FUNCTION_BLOCK RangeBasedPulse (* Distance based Impulse Generator *)
  (* Standard: 61499-1; Description: Copyright (c) 2025 HR Agrartechnik GmbH This program and the accompanying materials are made available under the terms of the Eclipse Public License 2.0 which is available at https://www.eclipse.org/legal/epl-2.0/ SPDX-License-Identifier: EPL-2.0 Distance based Impulse Generator START with a HIGH Pulse. *)
  (* Version 1.0, 2024-10-18, Franz Höpfinger, HR Agrartechnik GmbH, initial Version *)
  (* Version 1.1, 2024-10-18, Franz Höpfinger, HR Agrartechnik GmbH, added Offset *)
  PACKAGE signalprocessing::distance;
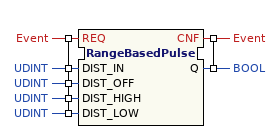
  EVENT_INPUT
    REQ WITH DIST_IN, DIST_OFF, DIST_HIGH, DIST_LOW; (* Normal Execution Request *)
  END_EVENT
  EVENT_OUTPUT
    CNF WITH Q; (* Execution Confirmation *)
  END_EVENT
  VAR_INPUT
    DIST_IN : UDINT; (* Travelled Distance *)
    DIST_OFF : UDINT; (* Distance Offset *)
    DIST_HIGH : UDINT; (* Distance for Output HIGH *)
    DIST_LOW : UDINT; (* Distance for Output LOW *)
  END_VAR
  VAR_OUTPUT
    Q : BOOL; (* Output *)
  END_VAR
  VAR
    DIST_REMAINDER : UDINT;
  END_VAR
  EC_STATES
    REQ : REQ -> CNF;
  END_STATES
  ALGORITHM REQ IN ST:
DIST_REMAINDER := (DIST_IN + DIST_OFF) MOD (DIST_HIGH + DIST_LOW);

Q := DIST_REMAINDER>= DIST_HIGH;
  END_ALGORITHM
END_FUNCTION_BLOCK
